(* Logix 5000 project; controller PracticaFlancos_set_reset Emulate 5570 rev 30.12; software revision 30.00 *)

TASK MainTask (continuous, watchdog 500 ms) : MainProgram

MODULES
   Local : Emulate 5570 (ICP 2, rev 30.12)
      I_O : vendor 1 type 0 code 15 (ICP 3, rev 1.1, Output RPI 150 ms)
END_MODULES

VAR_GLOBAL   (* controller tags *)
   FIO_Arranque : DINT;
   FIO_Auto : DINT;
   FIO_Banda1 : DINT;
   FIO_Banda2 : DINT;
   FIO_ESD : DINT;
   FIO_Fierro : DINT;
   FIO_KMI : DINT;
   FIO_Manual : DINT;
   FIO_Parada : DINT;
   FIO_Reset : DINT;
   FIO_Sensor1 : DINT;
   FIO_Sensor2 : DINT;
   FIO_Sensor3 : DINT;
END_VAR

PROGRAM MainProgram   (* main routine MainRoutine *)

ROUTINE MainRoutine   (* ladder *)
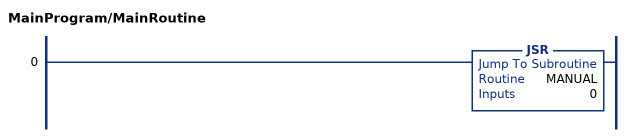
   0 (stored rung type 13): JSR(MANUAL,0);
END_ROUTINE

ROUTINE MANUAL   (* ladder *)
END_ROUTINE
END_PROGRAM
